KUKA KRL program: git_clean_demo.src, git_clean_demo.dat

--- git_clean_demo.src ---
&ACCESS RVP
&REL 48
&COMMENT WorkVisual Git Metadata Demonstration
&PARAM EDITMASK = *
&PARAM TEMPLATE = C:\KRC\Roboter\Template\vorgabe
DEF git_clean_demo()
  ; Use command: 'krl.cleanGitMetadata' to test stripping WorkVisual headers
  $OUT[1] = TRUE
END

--- git_clean_demo.dat ---
&ACCESS RVP
&REL 48
&COMMENT WorkVisual Header DAT
&PARAM EDITMASK = *
DEFDAT git_clean_demo
  DECL INT nVersion = 48
ENDDAT
